// TwinCAT 3 PLC project SafetyPLC
// ProgramVersion: 3.1.4026.19
// libraries:
//   Tc2_Standard, * (Beckhoff Automation GmbH)
//   Tc2_System, * (Beckhoff Automation GmbH)
//   Tc3_Module, * (Beckhoff Automation GmbH)
// project tree:
//   GVLs/ GVL_IO_SAFETY.TcGVL
//   / PlcTask.TcTTO
//   POUs/ MAIN.TcPOU, P_SAFETY.TcPOU
// (motion and I/O tree: see PLC project programplc)
// real-time tasks:
//   TASK MainTask: cycle T#3ms, priority 20, ADS port 350
//   TASK SafetyTask: cycle T#10ms, priority 22, ADS port 351
//   TASK WeightTask: cycle T#2ms, priority 19, ADS port 354
//   TASK PlcTask: cycle T#10ms, priority 21, ADS port 355
//   TASK TaskToRefreshEAP: cycle T#1ms, priority 12, ADS port 301
// variable links:
//   (this object) <-> SafetyPLC/SafetyPLC Instance
//     PlcTask Inputs/GVL_IO.IbBottleFeederSafety <-> PlcTask Outputs/GVL_IO_SAFETY.QbBottleFeederSafety
//     PlcTask Inputs/GVL_IO.IbCommunicationErrorUF50 <-> PlcTask Outputs/GVL_IO_SAFETY.QbCommunicationErrorUF50
//     PlcTask Inputs/GVL_IO.IbCommunicationErrorUP50B <-> PlcTask Outputs/GVL_IO_SAFETY.QbCommunicationErrorUP50B
//     PlcTask Inputs/GVL_IO.IbEmergencyStopButton <-> PlcTask Outputs/GVL_IO_SAFETY.QbEmergencyStopButton
//     PlcTask Inputs/GVL_IO.IbSafetyResetIn <-> PlcTask Outputs/GVL_IO_SAFETY.bSafetyResetOut
//     PlcTask Outputs/GVL_IO.QbSafetyResetBottleSorterIn <-> PlcTask Inputs/GVL_IO_SAFETY.IbSafetyResetBottleSorterIn
//     PlcTask Outputs/GVL_IO.QbSafetyResetCapSorterIn <-> PlcTask Inputs/GVL_IO_SAFETY.IbSafetyResetCapSorterIn
//     PlcTask Outputs/GVL_IO.QbSafetyResetDelay <-> PlcTask Inputs/GVL_IO_SAFETY.IbSafetyResetDelay
//     WeightTask Inputs/GVL_IO.IbEmergencyStop <-> PlcTask Outputs/GVL_IO_SAFETY.QbEmergencyStop

CONFIGURATION SafetyPLC
    RESOURCE PLC ON TwinCAT3
        TASK PlcTask(INTERVAL := T#10ms, PRIORITY := 22);
        PROGRAM MAIN WITH PlcTask : MAIN;
    END_RESOURCE
END_CONFIGURATION

// ---- GVLs/GVL_IO_SAFETY.TcGVL
VAR_GLOBAL
//15.10.2025 Vasyl dodanie sygnałów safety ze styków zasilania krokówek i Jiecang
	bErrorAck				AT %Q* :BOOL;	(* Potwierdzenie błędu *)
	bErrorAckGr2			AT %Q* :BOOL;	(* Potwierdzenie błędu UPB*)
	bErrorAckGr3			AT %Q* :BOOL;	(* Potwierdzenie błędu UF*)
	bSafetyResetIn 			AT %I* :BOOL;	//Przycisk resetu z panelu
	bSafetyResetInRC40		AT %I* :BOOL;	//Przycisk resetu z panelu
	
	bTurnTableSafetyResetIn AT %I* :BOOL;	//Przycisk resetu z panelu {warning 'dodać reset z turntable'}
	bPucksInserterSafetyResetIn AT %I* :BOOL;	//Przycisk resetu z panelu {warning 'dodać reset z turntable'}	
	bSafetyResetOut 		AT %Q* :BOOL;	//Info dla programu głównego	
	bSafetyReset 			AT %Q* :BOOL;
	bSafetyReset2 			AT %Q* :BOOL;
	bSafetyReset3			AT %Q* :BOOL; 
	bEmergencyStopButton 	AT %I* :BOOL; //Jeśli FALSE - Estop wysyołany przez przyciski
	bEmergencyStop 			AT %I* :BOOL; //Jeśli TRUE - maszyna w stanie bezpiecznym, FALSE - EStop
	bBottleFeederSafety		AT %I* :BOOL; // Status safety podajnika butelek
	bRobotEmergencyStop		AT %I* :BOOL; //Bezpieczeństwo robota 
	IbSafetyResetDelay	 	AT %I* :BOOL;	//Opóżnienie pierwszego zresetowania safety
	
	//Sygnały dla ProgramPLC
	QbEmergencyStopButton 	AT %Q* :BOOL; //Jeśli FALSE - Estop wysyołany przez przyciski
	QbEmergencyStop 		AT %Q* :BOOL; //Jeśli TRUE - maszyna w stanie bezpiecznym, FALSE - EStop
	QbBottleFeederSafety	AT %Q* :BOOL; // Jeśli TRUE - podajnik butelek w stanie bezpieczenym, FALSE- otwarte drzwi
	QbCommunicationErrorUF50	AT %Q* :BOOL;
	QbCommunicationErrorUP50B	AT %Q* :BOOL;
	
	QbRUN_STOP				AT %Q* :BOOL; //Jeśli FALSE - Estop wysyołany przez przyciski
	QbRUN_STOP_GR2			AT %Q* :BOOL; //Jeśli FALSE - Estop wysyołany przez przyciski
	QbRUN_STOP_GR3			AT %Q* :BOOL; //Jeśli FALSE - Estop wysyołany przez przyciski
	
	IbSafetyResetCapSorterIn 	AT %I*	: BOOL;			// Przycisk Reset
	IbSafetyResetBottleSorterIn AT %I*	: BOOL;			// Przycisk Reset

	IbSafetyRelayJiecang	 	AT %I* :BOOL;	
	IbSafetyRelayPneumatics	 	AT %I* :BOOL;
	IbSafetyRelayMotorsRobotA	AT %I* :BOOL;
	IbSafetyRelayMotorsRobotB	AT %I* :BOOL;
	IbSafetyRelayRC40	 		AT %I* :BOOL;	
	
	IbComErr_Gr2			AT %I* : BOOL;
	IbFBErr_Gr2				AT %I* : BOOL;
	IbOtherErr_Gr2			AT %I* : BOOL;
	IbOutErr_Gr2			AT %I* : BOOL;
	
	IbComErr_Gr3			AT %I* : BOOL;
	IbFBErr_Gr3				AT %I* : BOOL;
	IbOtherErr_Gr3			AT %I* : BOOL;
	IbOutErr_Gr3			AT %I* : BOOL;
	
	IbUP50BDeactivated		AT %I* : BOOL	:=TRUE;	//Status kluczyka deaktywacji safety
	IbUF50Deactivated		AT %I* : BOOL	:=TRUE;	//Status kluczyka deaktywacji safety
	
END_VAR

// ---- POUs/MAIN.TcPOU
PROGRAM MAIN
VAR

	bVISSafetyResetIn: BOOL;
END_VAR

(*
bSafetyReset:=bSafetyResetIn OR bVISSafetyResetIn;
bErrorAck:=bSafetyResetIn OR bVISSafetyResetIn;
bSafetyReset2:=bSafetyResetIn OR bVISSafetyResetIn;

*)
P_SAFETY();

//Sygnały dla ProgramPLC
QbEmergencyStopButton:=bEmergencyStopButton;
QbEmergencyStop:=bEmergencyStop;
QbBottleFeederSafety:=bBottleFeederSafety;
//Na potrzeby rygli
bSafetyResetOut :=	bSafetyResetIn OR bPucksInserterSafetyResetIn OR bSafetyResetInRC40;

END_PROGRAM

// ---- POUs/P_SAFETY.TcPOU
//==================================================================================================
//							Beckhoff Automation Poland
//									19.09.2017
// Procedura restartu - najpierw grupa, pozniej karta, na koncu bloki
// Uwaga - w przypadku bledu grupy, bledy karty nie sa widoczne jeszce przez chwile po resecie grupy.
// Dlatego dodane jest opoznienie
//	v1.0 	|| TC v 3.1.4022.2 || - pierwsza wersja
//==================================================================================================
PROGRAM P_SAFETY
VAR
	iStep						: INT;
	tonDelay					: TON;
	bDelayReq					: BOOL;
	tonDelay2: TON;
	tonDelay3: TON;
END_VAR

tonDelay.IN 								:= iStep = 10 OR iStep = 40;
tonDelay.PT									:= T#300MS;
tonDelay();

tonDelay2.IN								:= iStep = 20;
tonDelay2.PT								:= T#100MS;
tonDelay2();

tonDelay3.IN								:= iStep = 30;
tonDelay3.PT								:= T#3000MS;
tonDelay3();
//flagi błędu komunikacji
QbCommunicationErrorUP50B					:= (IbComErr_Gr2 OR IbFBErr_Gr2 OR IbOtherErr_Gr2 OR NOT IbOutErr_Gr2) AND NOT IbUP50BDeactivated;
QbCommunicationErrorUF50					:= (IbComErr_Gr3 OR IbFBErr_Gr3 OR IbOtherErr_Gr3 OR NOT IbOutErr_Gr3) AND NOT IbUF50Deactivated;




// Procedura
CASE iStep OF
	
	0: // Oczekiwanie na reset
	IF ((bSafetyResetIn OR IbSafetyResetCapSorterIn OR IbSafetyResetBottleSorterIn OR bPucksInserterSafetyResetIn OR bSafetyResetInRC40) AND
		NOT bEmergencyStop) AND IbSafetyResetDelay //Opóżnieni 30s z UBL tylko przy pierwszym uruchomieniu
	 	THEN
		QbRUN_STOP_GR2				R= IbComErr_Gr2 OR IbFBErr_Gr2 OR IbOtherErr_Gr2 OR NOT IbOutErr_Gr2;
		QbRUN_STOP_GR3				R= IbComErr_Gr3 OR IbFBErr_Gr3 OR IbOtherErr_Gr3 OR NOT IbOutErr_Gr3;
		iStep 						:= iStep + 10;
	END_IF
	
	10:	// Reset bledu grupy - jesli jest
		QbRUN_STOP					:= TRUE;
		//QbRUN_STOP_GR2				R= IbComErr_Gr2 OR IbFBErr_Gr2 OR IbOtherErr_Gr2 OR NOT IbOutErr_Gr2;
		//QbRUN_STOP_GR3				R= IbComErr_Gr3 OR IbFBErr_Gr3 OR IbOtherErr_Gr3 OR NOT IbOutErr_Gr3;
		IF tonDelay.Q THEN
			QbRUN_STOP							:= TRUE;
			QbRUN_STOP_GR2						:= TRUE;
			QbRUN_STOP_GR3						:= TRUE;
			bErrorAck							:= TRUE;
			bErrorAckGr2						:= TRUE;
			bErrorAckGr3						:= TRUE;
			bSafetyReset			:= TRUE;
			bSafetyReset2			:= TRUE;
			iStep 								:= iStep + 10;
		END_IF
	
	20: // Reset bledu karty AX5805 - jesli jest
		IF tonDelay2.Q THEN
			bErrorAck			:= FALSE;
			bErrorAckGr2			:= FALSE;
			bErrorAckGr3			:= FALSE;
			bSafetyReset			:= FALSE;
			bSafetyReset2			:= FALSE;
			bSafetyReset3			:= TRUE;
			iStep 					:= iStep + 10;	
		END_IF
	

	30:
		IF tonDelay3.Q THEN
			bSafetyReset			:= FALSE;
			bSafetyReset2			:= FALSE;
			bSafetyReset3			:= false;
			iStep 					:= iStep + 10;	
		END_IF
	
	40:
		IF tonDelay.Q THEN
			bSafetyReset3			:= FALSE;
			iStep	 				:= 0;
		END_IF
	
END_CASE

END_PROGRAM
